Omron Sysmac Studio project SPA_P7 (Sysmac Studio 1.23.0.14, StandardProject)

# Controller new_Controller_0: NX1P2-1040DT1 version 1.18
Task PrimaryTask (priority 4, period or condition 2000): Programa0

VAR_GLOBAL
    m1_avance : BOOL;  (* at BuiltInIO://cpu/#0/Output_Bit_01 *)
    m2 : BOOL;
    m1_retroceso : BOOL;  (* at BuiltInIO://cpu/#0/Output_Bit_02 *)
END_VAR

PROGRAM Programa0
VAR
    Marcha : BOOL;
    Paro : BOOL;
    Sentido : BOOL;
END_VAR
VAR_EXTERNAL
    m1_avance : BOOL;
    m1_retroceso : BOOL;
END_VAR
VAR
    _p1 : BOOL;
END_VAR

(* Section Sección0: ladder, written here as Structured Text *)

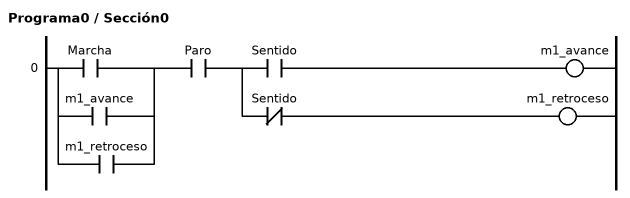
(* Rung 0 *)
_p1 := (Marcha OR m1_avance OR m1_retroceso) AND Paro;
m1_avance := (Marcha OR m1_avance OR m1_retroceso) AND Paro AND Sentido;
m1_retroceso := _p1 AND NOT Sentido;
END_PROGRAM